TYPE ST_CFG_DebugMsgManager :
STRUCT
	TCP_Driver		: ST_CFG_TcpDriver;
	SystemNumber	: INT;
END_STRUCT
END_TYPE

(* stored: Version 1.1.0.1, ProductVersion 3.1.4022.12
   DUT ST_CFG_DebugMsgManager: Id {0e629d44-6d36-4cec-9fd0-91195fd41f02} *)
